// TIA Portal V20 export
TYPE "typeCmHmiInterface"
// stored: Access Published, Namespace Unit1.Em13
   STRUCT
      softcam : "Unit1.Em13.typeCmHmiInterfaceSoftCam";
      brakeTest : "Unit1.Em13.typeCmHmiInterfaceBrakeTest";
   END_STRUCT;
END_TYPE
